{attribute addProperty BoxType "EJ3004-0000-0019"}
{attribute addProperty Id "UnderrangeBIT10.1251OverrangeBIT10.1252Limit_1_BIT_0BIT10.1253Limit_1_BIT_1BIT10.1253Limit_2_BIT_0BIT10.1255Limit_2_BIT_1BIT10.1255ErrorBIT10.1257TxPDO_StateBIT10.1257TxPDO_ToggleBIT10.1259"}
{attribute addProperty CRC "3338153583"}
{attribute addProperty SizeInBites "65"}
{attribute addProperty SizeInBytes "8.125"}
{warning 'Size of this structure is not a multiple of 8 bits!!!'}
TYPE Status_C6F82E6F :
STRUCT
	{attribute addProperty Name "Underrange"}
	Underrange : BIT;
	{attribute addProperty Name "Overrange"}
	Overrange : BIT;
	{attribute addProperty Name "Limit_1"}
	Limit_1_BIT_0 : BIT;
	{attribute addProperty Name "Limit_1"}
	Limit_1_BIT_1 : BIT;
	{attribute addProperty Name "Limit_2"}
	Limit_2_BIT_0 : BIT;
	{attribute addProperty Name "Limit_2"}
	Limit_2_BIT_1 : BIT;
	{attribute addProperty Name "Error"}
	Error : BIT;
	{attribute 'hide'}
	reserve_1 : BOOL;
	{attribute 'hide'}
	reserve_2_BOOL_0 : BOOL;
	{attribute 'hide'}
	reserve_2_BOOL_1 : BOOL;
	{attribute 'hide'}
	reserve_2_BOOL_2 : BOOL;
	{attribute 'hide'}
	reserve_2_BOOL_3 : BOOL;
	{attribute 'hide'}
	reserve_2_BOOL_4 : BOOL;
	{attribute 'hide'}
	reserve_2_BOOL_5 : BOOL;
	{attribute addProperty Name "TxPDO_State"}
	TxPDO_State : BIT;
	{attribute addProperty Name "TxPDO_Toggle"}
	TxPDO_Toggle : BIT;
END_STRUCT
END_TYPE

(* stored: Version 1.2.0.0, ProductVersion 3.1.4024.9
   DUT Status_C6F82E6F: Id {e1a265df-5e2f-4ce3-b360-ae544b7681e1} *)
